Universal Robots PolyScope program: 20240920_mediapipe.urp

Program 20240920_mediapipe (installation=20240827 directory=/programs/Demos/mediapipe createdIn=3.2.19275 lastSavedIn=5.15.1 robotSerialNumber=20245500285)
Calibrated DH parameters: a=[0.000097, -0.210459, -0.026602, 0.000137, 0.000078, 0]; d=[0.162601, 254.180657, -54.076236, -199.970743, 0.099615, 0.099684]; alpha=[1.569796, -0.001455, 0.001957, 1.570525, -1.571561, 0]; deltaTheta=[0, -1.053331, 8.839472, -1.50296, 0.000002, 0]
InitVariablesNode
BeforeStart
  MoveJ speed 50 deg/s, acceleration 40 deg/s^2 (useActiveTCP=true positionType=JointAngles) feature=Base
    Waypoint 路点_1: TCP in base x=83.397 y=-466.995 z=106.166 mm, rx=-2.2214 ry=-2.2214 rz=0.0001 rad; joints [83.677, -88.418, 117.225, -118.852, -90.036, 83.838] deg; TCP offset x=-0.17 y=0 z=192.95 mm, rx=0 ry=0 rz=0 rad
  joints := get_actual_joint_positions()
  SuppressedNode
    Halt
  home := get_actual_tcp_pose()
  Script: write_output_boolean_register(0, False )
  SuppressedNode
    Script: write_input_interger_register(0,0)
  Wait Sleep waitTime=0.01
  Script: popup("Registers reset, run PC code and then click Continue",title="Hi Daniel",blocking= True )
  mode := 0
Robot Program (runOnlyOnce=false)
  Script: write_output_boolean_register(0, True )
  Script: sync()
  Loop While (checkContinuously=false) expression=mode<3
    Loop While (checkContinuously=false) expression=mode≟1
      MoveJ speed 60 deg/s, acceleration 80 deg/s^2 (useActiveTCP=true) feature=Base
        Waypoint Variable (Variable): variable(name=joints)
      Script: write_output_boolean_register(0, False )
      Script: sync()
    Loop While (checkContinuously=false) expression=mode≟2
      Script: servoj(joints, 0, 0, 0.03, 0.9, 1800)
    Loop While (checkContinuously=false) expression=mode≟3
      Halt
  Script: sync()
Thread Thread_1 (runOnlyOnce=false)
  tmp := p[0,0,0,0,0,0]
  Loop Forever
    Script file /programs/pose_register.script
      | tmp[0]=read_input_float_register(0)
      | tmp[1]=read_input_float_register(1)
      | tmp[2]=read_input_float_register(2)
      | tmp[3]=read_input_float_register(3)
      | tmp[4]=read_input_float_register(4)
      | tmp[5]=read_input_float_register(5)
    joints := get_inverse_kin(p[tmp[0],tmp[1],tmp[2],tmp[3],tmp[4],tmp[5]],get_actual_joint_positions())
    Script: sync()
    mode := read_input_integer_register(0)
    Script: sync()
